(* IEC 61131-3 sources: CodesysTest/export/SX_1195.dev/Plc Logic/Application/PRJ Specific/1195 Testing/Clamping Mechanism/IClampingMechanism.itf, 2 files *)

(* ---- StartClamping.m.st ---- *)
(*#-#-#-#-#-#-#-#-#-#---Declaration---#-#-#-#-#-#-#-#-#-#-#-#-#*)

METHOD StartClamping : BOOL
VAR_INPUT
END_VAR

(* ---- StopClamping.m.st ---- *)
(*#-#-#-#-#-#-#-#-#-#---Declaration---#-#-#-#-#-#-#-#-#-#-#-#-#*)

METHOD StopClamping : BOOL
VAR_INPUT
END_VAR
